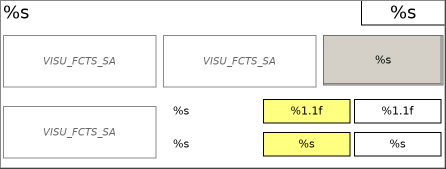
VISUALIZATION SA_LIGNE_GAZ_BROOKS_RAMPE  // 446x169
VAR_IN_OUT
	m_Input_Ligne:		BLOCK_LIGNE_GAZ;
	m_Input_Machine:	BLOCK_MODE_MARCHE_V2_0;
	m_Input_DG:			BLOCK_MFC_BROOKS_NoCoE;
	m_Input_UserRight:	BOOL;
END_VAR

VAR_INPUT
	m_Input_NumTextList:		INT;
END_VAR
    Rectangle (0,0 446x169), "%s", text list: 'TextList_Gaz', text index: m_Input_NumTextList
    Rectangle (361,0 85x25), "%s", text variable: m_Input_DG.CONF_Util_Name
    Frame (3,35 153x52)
        shows VISU_FCTS_SA(m_Input_ID_XML := 12, m_Input_UserRight := PRG_USER.ACTU_USER.FONCTION_SA AND NOT m_Input_Machine.STATE_Prod, m_Input_Operation := m_Input_Ligne.OP_MARCHE)
    Frame (3,106 153x52)
        shows VISU_FCTS_SA(m_Input_ID_XML := 13, m_Input_UserRight := PRG_USER.ACTU_USER.FONCTION_SA AND NOT m_Input_Machine.STATE_Prod, m_Input_Operation := m_Input_Ligne.OP_ARRET)
    Rectangle (170,99 91x24), "%s", text list: 'TextList_Gaz', text index: 3
    RoundedRectangle (354,99 87x24), "%1.1f", text variable: m_Input_DG.STATE_Flow
    RoundedRectangle (263,99 87x24), "%1.1f", text variable: m_Input_Ligne.PRM_Flow, input disabled if: (NOT PRG_USER.ACTU_USER.FONCTION_SA AND NOT m_Input_Machine.STATE_Prod) OR (NOT PRG_USER.ACTU_USER.MODIF_ENLIGNE AND m_Input_Machine.STATE_Prod)
        OnMouseClick: write the text variable via InputWithLimits, min 0, max m_Input_DG.CONF_Util_Max_Flow
    Rectangle (170,132 91x24), "%s", text list: 'TextList_Basiques', text index: 22
    RoundedRectangle (263,132 87x24), "%s", text variable: m_Input_Ligne.OP_RAMPE.PRM_Temps, input disabled if: (NOT PRG_USER.ACTU_USER.FONCTION_SA AND NOT m_Input_Machine.STATE_Prod) OR (NOT PRG_USER.ACTU_USER.MODIF_ENLIGNE AND m_Input_Machine.STATE_Prod)
        OnMouseClick: write the text variable via InputWithLimits
    Frame (163,35 153x52)
        shows VISU_FCTS_SA(m_Input_ID_XML := 14, m_Input_UserRight := PRG_USER.ACTU_USER.FONCTION_SA AND NOT m_Input_Machine.STATE_Prod, m_Input_Operation := m_Input_Ligne.OP_RAMPE.MARCHE)
    Button (323,35 120x50), "%s", input disabled if: (NOT PRG_USER.ACTU_USER.FONCTION_SA AND NOT m_Input_Machine.STATE_Prod) OR (NOT PRG_USER.ACTU_USER.MODIF_ENLIGNE AND m_Input_Machine.STATE_Prod), text list: 'TextList_Basiques', text index: 19
        toggle m_Input_Ligne.CO_Modif
    RoundedRectangle (354,132 87x24), "%s", text variable: m_Input_Ligne.OP_RAMPE.OUT_Tps_ecoule
END_VISUALIZATION

(* stored: Version 1.1.0.1, ProductVersion 3.1.4024.10
   Visu SA_LIGNE_GAZ_BROOKS_RAMPE: Id {99d91c14-562b-4d90-a3a2-f91106485f65} *)
